Staubli VAL3: link_all.pgx

public program link_all(string x_sName)
  local num i
begin
  // link all
  link(tTraj[x_sName].fFrame,world)
  tTraj[x_sName].fFrame.trsf=saveData:fFrameItem[tTraj[x_sName].nIndexFrame].fFrame.trsf
  for i=0 to size(tTraj[x_sName].tData)-1
    link(tTraj[x_sName].tData[i].pPoint,tTraj[x_sName].fFrame)
  endFor
end
